TYPE CyclicAxis_monitor_typ :
STRUCT
END_STRUCT
END_TYPE

(* stored: Version 1.1.0.1, ProductVersion 3.1.4024.3
   DUT CyclicAxis_monitor_typ: Id {355b4888-da76-0250-21d7-28c4211ba016} *)
